TYPE ST_EndurancePyrometerErrorResponse :
STRUCT
	Code	: Tc2_System.T_MaxString;
	Message	: STRING;
END_STRUCT
END_TYPE

(* stored: Version 1.1.0.1, ProductVersion 3.1.4024.16
   DUT ST_EndurancePyrometerErrorResponse: Id {44305f1c-1a9e-0507-18c4-34e5b47762e3} *)
